RoboDK station: Simulation copy.rdk

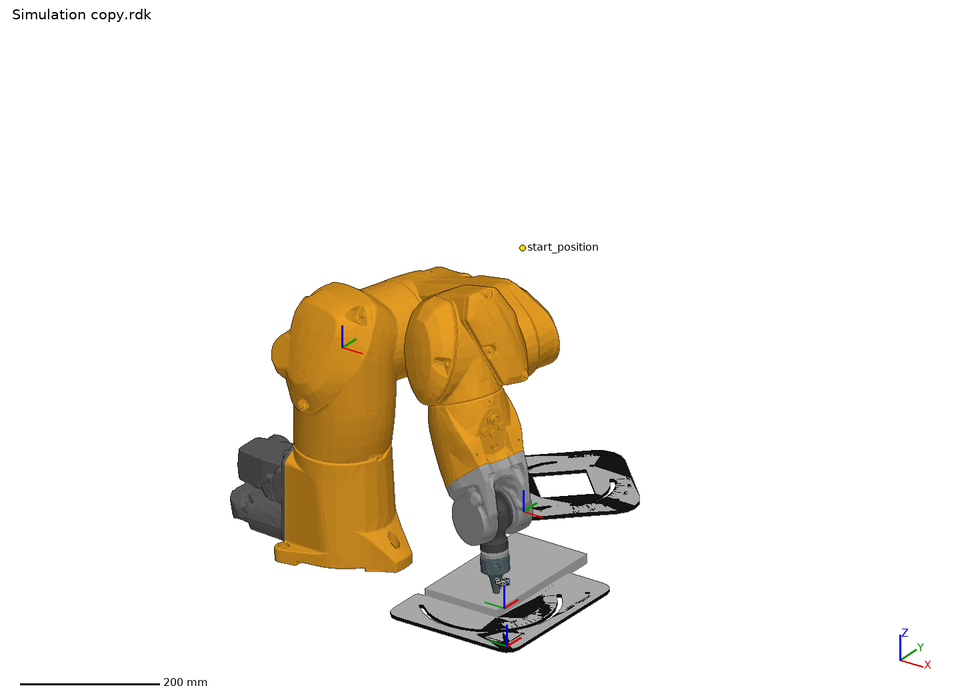
[picture v0: the station drawn from its stored meshes, robots at their saved joint values, targets as dots, program paths as lines]
Station Simulation (saved by RoboDK 5.9.1). Poses are relative to the parent item; angles as X-Y-Z fixed-axis rotations.
  - frame Staubli TX2-40 Base at (0, 0, 0) mm
    - robot Staubli TX2-40: 6 axes, payload 2 kg, reach 515 mm, repeatability 0.02 mm, weight 29 kg
        modified DH rows (alpha deg, a mm, theta deg, d mm): 0, 0, 0, 320; -90, 0, -90, 35; 0, 225, -90, 0; -90, 0, 0, 225; 90, 0, 0, 0; -90, 0, 180, 65
        base shift (0, 0, -320) mm
        joint limits [-180, -125, -138, -270, -120, -270] to [180, 125, 138, 270, 133.5, 270]; home [0, 0, 90, 0, 0, 0]; saved at [-16.064, 76.951, 82.635, 0, 15.97, -16.064]
      - tool AROB_LWS_VakuumGreifer_14, TCP at (0, 0, 0) mm, size 81.8 x 41.9 x 49.7 mm, geometry from AROB_LWS_VakuumGreifer_14.stp
    - target start_position (Cartesian target) at (290, 35, 225) mm, rotated rx 0 ry 90 rz 0 deg; joints [0, 0, 90, 0, 0, 0] of Staubli TX2-40
    - target idle_position (Cartesian target) at (290, 35, 225) mm, rotated rx 0 ry 90 rz 0 deg; joints [0, 0, 90, 0, 0, 0] of Staubli TX2-40
    - target home_position (Cartesian target) at (290, 35, 225) mm, rotated rx 0 ry 90 rz 0 deg; joints [0, 0, 90, 0, 0, 0] of Staubli TX2-40
  - frame MagazineFrame at (400, -160, -300) mm, rotated rx 0 ry 0 rz 90 deg
    - object AROB_Magazinplatte at (100, 100, 0) mm, size 260 x 220 x 5 mm, geometry from AROB_Magazinplatte.stl
    - frame JengaPieces at (100, 75, 0) mm
      - object AROB_Jengastuck1 at (0, 0, 0) mm, size 75 x 25 x 15 mm, geometry from AROB_Jengastuck.stl
      - object AROB_Jengastuck2 at (0, 25, 0) mm, size 75 x 25 x 15 mm, geometry from AROB_Jengastuck.stl
      - object AROB_Jengastuck3 at (0, 50, 0) mm, size 75 x 25 x 15 mm, geometry from AROB_Jengastuck.stl
      - object AROB_Jengastuck4 at (0, 75, 0) mm, size 75 x 25 x 15 mm, geometry from AROB_Jengastuck.stl
      - object AROB_Jengastuck5 at (0, 100, 0) mm, size 75 x 25 x 15 mm, geometry from AROB_Jengastuck.stl
      - object AROB_Jengastuck6 at (75, 0, 0) mm, size 75 x 25 x 15 mm, geometry from AROB_Jengastuck.stl
      - object AROB_Jengastuck7 at (75, 25, 0) mm, size 75 x 25 x 15 mm, geometry from AROB_Jengastuck.stl
      - object AROB_Jengastuck8 at (75, 50, 0) mm, size 75 x 25 x 15 mm, geometry from AROB_Jengastuck.stl
      - object AROB_Jengastuck9 at (75, 75, 0) mm, size 75 x 25 x 15 mm, geometry from AROB_Jengastuck.stl
      - object AROB_Jengastuck10 at (75, 100, 0) mm, size 75 x 25 x 15 mm, geometry from AROB_Jengastuck.stl
      - object AROB_Jengastuck11 at (150, 0, 0) mm, size 75 x 25 x 15 mm, geometry from AROB_Jengastuck.stl
      - object AROB_Jengastuck12 at (150, 25, 0) mm, size 75 x 25 x 15 mm, geometry from AROB_Jengastuck.stl
      - object AROB_Jengastuck13 at (150, 50, 0) mm, size 75 x 25 x 15 mm, geometry from AROB_Jengastuck.stl
      - object AROB_Jengastuck14 at (150, 75, 0) mm, size 75 x 25 x 15 mm, geometry from AROB_Jengastuck.stl
      - object AROB_Jengastuck15 at (150, 100, 0) mm, size 75 x 25 x 15 mm, geometry from AROB_Jengastuck.stl
  - frame TowerFrame at (120, 280, -340) mm
    - object AROB_Turmplatte at (0, 100, 0) mm, rotated rx 0 ry 0 rz 45 deg, size 200 x 200 x 5 mm, geometry from AROB_Turmplatte.stl
  - Python program main (listed below)

--- Python program main ---
from magazine import Magazine
from tower import Tower
from robot_controller import RobotController

def main():
    mag = Magazine()
    tower = Tower()
    robot = RobotController()

    robot.move_to_home()

    for i in range(15):
        print(f"Handling Block {i+1}")
        pick_pose = mag.next_pick_pose()
        place_pose = tower.next_place_pose()

        robot.pick(pick_pose)
        robot.move_to_home()
        robot.place(place_pose)
        robot.move_to_home()

    print("Jenga-Turm erfolgreich aufgebaut.")
    robot.move_to_home()

if __name__ == "__main__":
    main()
